// TIA Portal V17 export
// export: Created 2025-03-12T14:52:43.8164211Z, ExportSetting WithDefaults, DisplayName Totally Integrated Automation Portal, DisplayVersion V17 Update 8, DisplayName TIA Portal Openness, DisplayVersion V17 Update 8, DisplayName TIA Portal Version Control Interface, DisplayVersion V17, DisplayName SINAMICS Startdrive Advanced, DisplayVersion V17 SP2, DisplayName SINAMICS Startdrive G110M, G120, G120C, G120D, G120P, G115D, DisplayVersion V17 SP2, DisplayName SINAMICS Startdrive G130, G150, S120, S150, SINAMICS MV, S210, DisplayVersion V17 SP2, DisplayName STEP 7 Professional, DisplayVersion V17 Update 8, DisplayName SINUMERIK ONE STEP 7 Toolbox, DisplayVersion V17 Update 12, DisplayName SINUMERIK 840D sl STEP 7 Toolbox, DisplayVersion V17 Update 12, DisplayName STEP 7 Safety, DisplayVersion V17 Update 6, DisplayName WinCC Advanced, DisplayVersion V17 Update 8
TYPE "UDT_Feeder Line"
// stored: IsFailsafeCompliant false
   STRUCT
      GAS_FLOW_RATE_ACTUAL : Real;   // GAS FLOW RATE - ACTUAL
      GAS_FLOW_RATE_AUTO : Real;   // GAS FLOW RATE - AUTO
      GAS_FLOW_RATE_MANUAL : Real;   // GAS FLOW RATE - MANUAL
      DISC_SPEED_ACTUAL : Real;   // DISC SPEED - ACTUAL
      DISC_SPEED_AUTO : Real;   // DISC SPEED - AUTO
      DISC_SPEED_MANUAL : Real;   // DISC SPEED - MANUAL
      STIRRER_SPEED_ACTUAL : Real;   // STIRRER SPEED - ACTUAL
      STIRRER_SPEED_AUTO : Real;   // STIRRER SPEED - AUTO
      STIRRER_SPEED_MANUAL : Real;   // STIRRER SPEED - MANUAL
      HOPPER_TEMP_ACTUAL : Real;   // HOPPER TEMP - ACTUAL
      HOPPER_TEMP_AUTO : Real;   // HOPPER TEMP - AUTO
      HOPPER_TEMP_MANUAL : Real;   // HOPPER TEMP - MANUAL
      HEATER_ON_MANUAL_REQUEST : Bool;   // HEATER ON MANUAL REQUEST
      HEATER_OFF_MANUAL_REQUEST : Bool;   // HEATER OFF MANUAL REQUEST
      HEATER_STATUS : Byte;   // HEATER STATUS
      HOPPER_ON_MANUAL_REQUEST : Bool;   // HOPPER ON MANUAL REQUEST
      HOPPER_OFF_MANUAL_REQUEST : Bool;   // HOPPER OFF MANUAL REQUEST
      HOPPER_STATUS : Byte;   // HOPPER STATUS
      START_SEQUENCE_GAS_STEPS : Int;   // START SEQUENCE GAS STEPS
      START_SEQUENCE_DISK_STEPS : Int;   // START SEQUENCE DISK STEPS
      STOP_SEQUENCE_GAS_STEPS : Int;   // STOP SEQUENCE GAS STEPS
      STOP_SEQUENCE_DISK_STEPS : Int;   // STOP SEQUENCE DISK STEPS
      STOP_SEQUENCE_PAUSE_STEP : Int;   // STOP SEQUENCE PAUSE STEP
      DISC_SPEED_WARNING_UPPER_LIMIT : Real;   // DISC SPEED - WARNING UPPER LIMIT
      DISC_SPEED_ALARM_UPPER_LIMIT : Real;   // DISC SPEED - ALARM UPPER LIMIT
      DISC_SPEED_WARNING_LOWER_LIMIT : Real;   // DISC SPEED - WARNING LOWER LIMIT
      DISC_SPEED_ALARM_LOWER_LIMIT : Real;   // DISC SPEED - ALARM LOWER LIMIT
      GAS_FLOW_RATE_WARNING_UPPER_LIMIT : Real;   // GAS FLOW RATE - WARNING UPPER LIMIT
      GAS_FLOW_RATE_ALARM_UPPER_LIMIT : Real;   // GAS FLOW RATE - ALARM UPPER LIMIT
      GAS_FLOW_RATE_WARNING_LOWER_LIMIT : Real;   // GAS FLOW RATE - WARNING LOWER LIMIT
      GAS_FLOW_RATE_ALARM_LOWER_LIMIT : Real;   // GAS FLOW RATE - ALARM LOWER LIMIT
      STIRRER_SPEED_WARNING_UPPER_LIMIT : Real;   // STIRRER SPEED - WARNING UPPER LIMIT
      STIRRER_SPEED_ALARM_UPPER_LIMIT : Real;   // STIRRER SPEED - ALARM UPPER LIMIT
      STIRRER_SPEED_WARNING_LOWER_LIMIT : Real;   // STIRRER SPEED - WARNING LOWER LIMIT
      STIRRER_SPEED_ALARM_LOWER_LIMIT : Real;   // STIRRER SPEED - ALARM LOWER LIMIT
      HOPPER_TEMP_ALARM_UPPER_LIMIT : Real;   // HOPPER TEMP - ALARM UPPER LIMIT
      PRESSURE_VALUE_CURRENT_SENSOR : Real;   // PRESSURE VALUE - CURRENT SENSOR
   END_STRUCT;
END_TYPE
